// Core §2.7 — quality bit stored with every generated wall-clock record.
FUNCTION F_TimeSynchronized : BOOL

F_TimeSynchronized := GVL_FraktalTime.Current.Available
    AND GVL_FraktalTime.Current.Synchronized;

END_FUNCTION

(* stored: Version 1.1.0.1, ProductVersion 3.1.4024.12
   POU F_TimeSynchronized: Id {e3d213ce-3d17-457a-9d41-f429026717b5}, SpecialFunc None *)
